PROGRAM FB_PBR260
VAR
	AO:INT;
	rPRESS:REAL;
	xPRESS_OK:BOOL;
	xHV_DIS:BOOL;
END_VAR

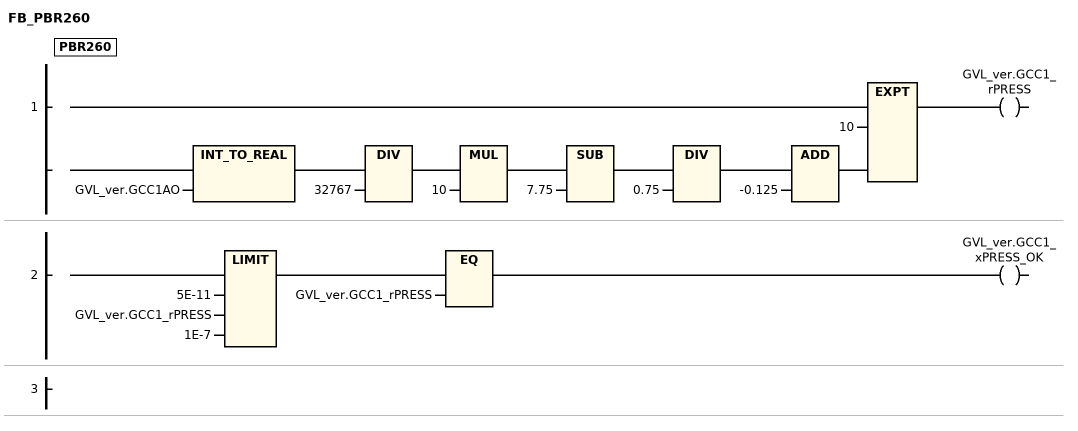
// NETWORK 1
PBR260:
GVL_ver.GCC1_rPRESS := EXPT(10, ((INT_TO_REAL(GVL_ver.GCC1AO) / 32767) * 10 - 7.75) / 0.75 + -0.125);

// NETWORK 2
GVL_ver.GCC1_xPRESS_OK := LIMIT(5E-11, GVL_ver.GCC1_rPRESS, 1E-7) = GVL_ver.GCC1_rPRESS;

// NETWORK 3

END_PROGRAM

(* stored: Version 1.1.0.1, ProductVersion 3.1.4022.3
   POU FB_PBR260: Id {79cc6bf8-793a-40e8-901a-d5be14f7d3c8}, SpecialFunc None *)
